PROGRAM Visu
VAR
	bStartTL1 : BOOL;
	bStartTL2 : BOOL;
	bStartTL3 : BOOL;
END_VAR

END_PROGRAM

(* stored: Version 1.1.0.1, ProductVersion 3.1.4024.2
   POU Visu: Id {2c780e66-9945-423c-a677-d03b9608941b}, SpecialFunc None *)
